FUNCTION_BLOCK ValueBuffer
VAR_INPUT
	fValue : REAL;
END_VAR
VAR
	values: ARRAY[0 .. globals.MAX_BUFFER_LENGTH] OF REAL;
	bInitialized: BOOL:=FALSE;
	nStoreEveryNthValue : UINT:=1;
	nCurrentIndex : UDINT:=1;
	eBufState : BufferState:=BufferState.INIT;
	nBufSize : UDINT:=1000;
	nTickCount : UDINT;
END_VAR

IF NOT bInitialized THEN
	// removed: dynamic memory allocation
	// reason: couldn't find a way to read via pyads (Error 1793 "Service is not supported by server")
	bInitialized := TRUE;
	eBufState := BufferState.IDLE;
END_IF

StoreValueConditional(fValue);

METHOD PUBLIC PrepareBuffer
VAR_INPUT
	nNumValues: UDINT;
END_VAR
VAR_OUTPUT
	nNumPrepared: UDINT;
END_VAR
VAR
	n: UDINT;
END_VAR
IF eBufState = BufferState.IDLE OR eBufState = BufferState.FULL THEN
	// IF nNumValues <> nBufSize THEN
		// fbMemoryBuffer.Resize(nSize:=nNumValues * SIZEOF(REAL), bPreserve:=FALSE, bReset:=TRUE);
		// values := fbMemoryBuffer.pBuffer;
		// nBufSize := nNumValues;
	// ELSE
		// fbMemoryBuffer.Clear();
	// END_IF
	nBufSize := MIN(nNumValues, globals.MAX_BUFFER_LENGTH);
	nNumPrepared := nBufSize;
	FOR n := 0 TO nBufSize DO
		values[n] := 0;
	END_FOR
eBufState := BufferState.IDLE;
nCurrentIndex := 0;
nTickCount := 0;
END_IF
END_METHOD

METHOD StartBuffer
IF eBufState = BufferState.IDLE THEN
	eBufState := BufferState.STORING;
END_IF
END_METHOD

METHOD StopBuffer
eBufState := BufferState.FULL;
END_METHOD

METHOD StoreValueConditional // Store value in buffer if tick count MOD buffer rate equals 0 
VAR_INPUT
	fValue : REAL;
END_VAR
IF eBufState = BufferState.STORING THEN
	IF (nTickCount MOD nStoreEveryNthValue) = 0 THEN
		values[nCurrentIndex] := fValue;
		nCurrentIndex := nCurrentIndex + 1;
	END_IF
	nTickCount := nTickCount + 1;
END_IF

IF nCurrentIndex >= nBufSize OR nCurrentIndex >= globals.MAX_BUFFER_LENGTH THEN
	eBufState := BufferState.FULL;
END_IF
END_METHOD

END_FUNCTION_BLOCK

(* stored: Version 1.1.0.1, ProductVersion 3.1.4024.12
   POU ValueBuffer: Id {36de9085-401e-4161-a47c-a7ed199b0f9f}, SpecialFunc None
   Method PrepareBuffer: Id {cfacde04-1779-43c7-b4e4-baead0d51989}
   Method StartBuffer: Id {1251b1d5-52c8-4328-8a8e-b4d9070eeefc}
   Method StopBuffer: Id {069f8ae3-41d5-4395-b5eb-26835483a8f2}
   Method StoreValueConditional: Id {46265f77-403d-4aa2-9c61-79688ea47cf2} *)
